Staubli VAL3: start.pgx

program start()
begin
  // Se pone en marcha la aplicacion

  // Se establece el valor inicial de variables globales
  // BOOL
  bPiezaPreparada=false
  bFin=false
  bTermina=false
  bTraslada=false

  // NUM
  nSolicitadas=1
  nPendientes=0

  // STRING
  sMensaje=""

  // Se crean e inician las tareas de la aplicacion
  taskCreate "mcp",100,mcp()
  taskCreate "robot",100,robot()
end
